# B&R Automation Studio project TD52 (part 38)

#### AdditionalFunctions.st - Additional functions
```iecst
(*******************************************************************************
coupling        additional functions

This code is confidential and proprietary to the INNIO Company.
It may not be used in any form, or reproduced in any manner,
without written permission of the INNIO Company.
Copyright, INNIO Company, 2019

Customized modifications: -
------------------------

History:
-------
V0.00.0	17.07.2012	froehlichw	new
V0.00.1	14.01.2019	Denk		adapted for bus test forcing

Instructions for use:
--------------------

Outstandings:
------------

(*******************************************************************************)

(*-----------------------------------------------------------------
/* compress and copy BOOL-Array at scrAdr to INT-Array at dstAdr
/* IN: scrAdr ... source address (start address of BOOL-Array)
/*     dstAdr ... destination address (base address=[0] of INT-Array)
/*     idxMin ... start index of INT-Array for copy
/*     idxMax ... end index of INT-Array for copy
/*---------------------------------------------------------------*)
ACTION BusTest_BOOL_TO_INT:
	FOR idx1:= idxMin TO idxMax DO
		pScrData ACCESS (srcAdr + (idx1 - idxMin) * 16);
		pDstData ACCESS (dstAdr + SIZEOF(pDstData) * idx1);
		pDstData.0:= pScrData[0];
		pDstData.1:= pScrData[1];
		pDstData.2:= pScrData[2];
		pDstData.3:= pScrData[3];
		pDstData.4:= pScrData[4];
		pDstData.5:= pScrData[5];
		pDstData.6:= pScrData[6];
		pDstData.7:= pScrData[7];
		pDstData.8:= pScrData[8];
		pDstData.9:= pScrData[9];
		pDstData.10:= pScrData[10];
		pDstData.11:= pScrData[11];
		pDstData.12:= pScrData[12];
		pDstData.13:= pScrData[13];
		pDstData.14:= pScrData[14];
		pDstData.15:= pScrData[15];
	END_FOR;
END_ACTION

(*-----------------------------------------------------------------
/* compress AND copy INT-Array at srcAdr TO BOOL-Array at dstAdr
/* IN: dstAdr ... destination address (start address OF BOOL-Array)
/*     scrAdr ... source address (base address=[0] OF INT-Array)
/*     idxMin ... start index OF INT-Array FOR copy
/*     idxMax ... end index OF INT-Array FOR copy
/*---------------------------------------------------------------*)
ACTION BusTest_INT_TO_BOOL:
	FOR idx1:= idxMin TO idxMax DO
		pScrData1 ACCESS (srcAdr + SIZEOF(pScrData1) * idx1);
		pDstData1 ACCESS (dstAdr + (idx1 - idxMin) * 16);
		pDstData1[0]:= pScrData1.0;
		pDstData1[1]:= pScrData1.1;
		pDstData1[2]:= pScrData1.2;
		pDstData1[3]:= pScrData1.3;
		pDstData1[4]:= pScrData1.4;
		pDstData1[5]:= pScrData1.5;
		pDstData1[6]:= pScrData1.6;
		pDstData1[7]:= pScrData1.7;
		pDstData1[8]:= pScrData1.8;
		pDstData1[9]:= pScrData1.9;
		pDstData1[10]:= pScrData1.10;
		pDstData1[11]:= pScrData1.11;
		pDstData1[12]:= pScrData1.12;
		pDstData1[13]:= pScrData1.13;
		pDstData1[14]:= pScrData1.14;
		pDstData1[15]:= pScrData1.15;
	END_FOR;
END_ACTION
```

#### coupling.var - Local variables
```iecst
VAR
	ucTeilerLauf : USINT; (* TK4 splitter variable *)
	ucINIT : ARRAY[0..1] OF USINT; (* initialise all coupling types *)
	szMode1 : STRING[50]; (* string interface mode 1 *)
	szInterface05 : STRING[40]; (* string interface 5 *)
	szInterface04 : STRING[40]; (* string interface 4 *)
	szInterface03 : STRING[40]; (* string interface 3 *)
	szInterface02_Comm2 : STRING[40]; (*Profibus communication2, slave2 *)
	szInterface02_Comm1 : STRING[40]; (*Profibus communication1, slave2 *)
	szInterface02 : STRING[40]; (* string interface 2 *)
	szInterface01_Comm2_PN : STRING[40]; (*Profinet communication2, slave1*)
	szInterface01_Comm2 : STRING[40]; (*Profibus communication2, slave1 *)
	szInterface01_Comm1_PN : STRING[40]; (*Profinet communication1, slave1 *)
	szInterface01_Comm1 : STRING[40]; (*Profibus communication1, slave1 *)
	szInterface01 : STRING[40]; (* string interface 1 *)
	szHilf1 : STRING[50]; (* help sting 1 *)
	szDevice1 : STRING[40]; (* string interface position 1 *)
	StationNumber : STRING[3];
	StationName1 : STRING[30] := ''; (*Profinet communication 1, station name*)
	Station : UDINT;
	Start_PN_Slave1 : USINT; (*Index variable*)
	Start_PB_Slave2 : USINT; (*Index variable*)
	Start_PB_Slave1 : USINT; (*Index variable*)
	siComm2_type : INT; (* couple type 2 old *)
	siComm2_Stopbit : INT; (* stop bits old Modbus *)
	siComm2_SlaveID : INT; (* ident for Modbus connection *)
	siComm2_Parity : INT; (* parity old Modbus *)
	siComm2_Interface : INT; (* position interface coupling 2 *)
	siComm2_Baud : INT; (* baudrate old Modbus *)
	siComm1_type : INT; (* couple type 1 old *)
	siComm1_Stopbit : INT; (* stop bits old Modbus *)
	siComm1_SlaveID : INT; (* ident for Modbus connection *)
	siComm1_Parity : INT; (* parity old Modbus *)
	siComm1_Interface : INT; (* position interface coupling 1 *)
	siComm1_Baud : INT; (* baudrate old Modbus *)
	nxpnsStartBusComm_01 : nxpnsStartBusComm;
	nxpnsSetName_01 : nxpnsSetName;
	nxdpsStartBusComm_02 : nxdpsStartBusComm;
	nxdpsStartBusComm_01 : nxdpsStartBusComm;
	nxdpsSetAdr_02 : nxdpsSetAdr;
	nxdpsSetAdr_01 : nxdpsSetAdr;
	MBT_4_2 : ARRAY[0..MODBUS_TCP_MAX_ARRAY] OF UINT := [MODBUS_TCP_MAX_ARRAY+1(0)]; (* data array Modbus TCP Coupling 2*)
	MBT_4_1 : ARRAY[0..MODBUS_TCP_MAX_ARRAY] OF UINT := [MODBUS_TCP_MAX_ARRAY+1(0)]; (* data array Modbus TCP Coupling 1*)
	MBSOpen_Var : ARRAY[0..1] OF MBSOpen; (* FUB Modbus open *)
	MBSlave_Var : ARRAY[0..1] OF MBSlave; (* FUB Modbus slave *)
	MBSClose_Var : ARRAY[0..1] OF MBSClose; (* FUB Modbus close *)
	MBR_4_2 : ARRAY[0..MODBUS_RTU_MAX_ARRAY] OF UINT := [MODBUS_RTU_MAX_ARRAY+1(0)]; (* data array Modbus RTU coupling 2 *)
	MBR_4_1 : ARRAY[0..MODBUS_RTU_MAX_ARRAY] OF UINT := [MODBUS_RTU_MAX_ARRAY+1(0)]; (* data array Modbus RTU coupling 1 *)
	MBinitOK : ARRAY[0..1] OF BOOL; (* initialising Modbus O.K. *)
	logErrorStringPN : STRING[100] := 'Error PROFINET communication slave 1';
	logErrorString2 : STRING[100] := 'Error PROFIBUS communication slave 2';
	logErrorStringModTCP : STRING[100] := 'Error MODBUS TCP set IP adress / Subnet mask slave';
	logErrorString1 : STRING[100] := 'Error PROFIBUS communication slave 1';
END_VAR
VAR CONSTANT
	IF4_IDLE : UINT := 0; (*Set IP adress and subnet mask IF4.ETH*)
	IP_IF4_SET : UINT := 1; (*Set IP adress IF4.ETH*)
	SUBMASK_IF4_SET : UINT := 2; (*Set Subnet mask IF4.ETH*)
	IF4_OK : UINT := 3; (*Set IP adress and subnet mask IF4.ETH OK*)
	OPEN_MODTCP : UINT := 4; (*Open Modbus TCP Communication*)
	IF4_ERR : UINT := 5; (*Set IP adress IF4.ETH Error*)
	PROFIBUS_MAX_RECV_2SLAVES : UINT := 16; (* max send data words profibus *)
	PROFIBUS_MAX_SEND_2SLAVES : UINT := 192; (* max send data words profibus *)
END_VAR
VAR
	iInterface02_Comm1 : UDINT; (*Adress Profibus Interface1, communication1, slave2*)
	iInterface01_Comm1_PN : UDINT; (*Adress Profinet Interface1, communication1, slave1*)
	iInterface01_Comm1 : UDINT; (*Adress Profibus Interface1, communication1, slave1 *)
	idx : INT;
	iComm1_PN_SlaveID1_old : INT; (*Profinet communication1, slave1 old adress*)
	iComm2_PN_SlaveID1_old : INT; (*Profinet communication1, slave1 old adress*)
	iComm1_PB_SlaveID1_old : INT; (*Profibus communication1, slave1 old adress*)
	iComm1_PB_SlaveID2_old : INT; (*Profibus communication1, slave2 old adress*)
	iComm2_PB_SlaveID1_old : INT; (*Profibus communication1, slave1 old adress*)
	iComm2_PB_SlaveID2_old : INT; (*Profibus communication1, slave2 old adress*)
	iComm_PB_SlaveID1 : INT; (*Profibus communication1, slave1 old adress*)
	iComm_PB_SlaveID2 : INT; (*Profibus communication1, slave1 old adress*)
	iComm_PN_SlaveID1 : INT; (*Profibus communication1, slave1 old adress*)
	AsArLogWrite_PN_01 : AsArLogWrite;
	AsArLogWrite_PB_02 : AsArLogWrite;
	AsArLogWrite_TCP : AsArLogWrite;
	AsArLogWrite_PB_01 : AsArLogWrite;
	AsArLogGetInfo_PN_01 : AsArLogGetInfo;
	AsArLogGetInfo_PB_02 : AsArLogGetInfo;
	AsArLogGetInfo_TCP : AsArLogGetInfo;
	AsArLogGetInfo_PB_01 : AsArLogGetInfo;
	InDataSwap : ARRAY[0..MAX_IN_DATA_ARRAY] OF INT;
	OutDataSwap : ARRAY[0..MAX_OUT_DATA_ARRAY] OF INT;
	OutDataOldSwap : ARRAY[0..MAX_OUT_DATA_ARRAY] OF INT;
	ArrayCntIn : INT;
	ArrayCntOut : INT;
	iStartRecvReg : INT;
	iStartRecvReg_old : INT;
	iStartSendReg : INT;
	iStartSendReg_old : INT;
	iIdx_Comm1_type_old : INT; (*Type of coupling 1 old, for detection of parameter change*)
	iIdx_Comm2_type_old : INT; (*Type of coupling 2 old, for detection of parameter change*)
	iBC_Test_Recv_Reg_old : ARRAY[0..MAX_IN_DATA_ARRAY_BUSTEST] OF INT;
	bBC_Test_Recv_Reg_old : ARRAY[0..MAX_IN_DATA_ARRAY_BOOL] OF BOOL;
	idx1 : INT;
	srcAdr : UDINT;
	dstAdr : UDINT;
	idxMin : INT;
	idxMax : INT;
	pScrData : REFERENCE TO ARRAY[0..15] OF BOOL;
	pDstData : REFERENCE TO UINT;
	pScrData1 : REFERENCE TO UINT;
	pDstData1 : REFERENCE TO ARRAY[0..15] OF BOOL;
	RegOffset_Send : INT;
	RegOffset_Recv : INT;
	xTON_BC_Test_Force_Active : TON;
	bBC_Test_Recv_Reg_Forced : ARRAY[0..MAX_IN_DATA_ARRAY] OF BOOL;
	bBC_Test_Send_Reg_Forced : ARRAY[0..MAX_OUT_DATA_ARRAY] OF BOOL;
	iBC_Test_Recv_Start_Reg_old : INT;
	iBC_Test_Send_Start_Reg_old : INT;
	bBC_Test_Recv_Reg_Forced_old : ARRAY[0..20] OF BOOL;
	bBC_Test_Send_Reg_Forced_old : ARRAY[0..20] OF BOOL;
	bBC_Test_Recv_Reg_AllForced : BOOL;
	bBC_Test_Send_Reg_AllForced : BOOL;
	bBC_Test_Recv_Reg_AllUnforced : BOOL;
	bBC_Test_Send_Reg_AllUnforced : BOOL;
	bBC_Test_Send_DW : BOOL; (*Dataword convention for send (Profibus, Profinet)*)
	iBC_Test_Send_DW : INT; (*Dataword convention for send (Profibus, Profinet)*)
	bBC_Test_Recv_DW : BOOL; (*Dataword convention for receive (Profibus, Profinet)*)
	iBC_Test_Recv_DW : INT; (*Dataword convention for receive (Profibus, Profinet)*)
	r : INT;
	i : INT;
	k : INT;
	t : INT;
	m : INT;
	n : INT;
	p : INT;
	v : INT;
	w : INT;
	x : INT;
	b : INT;
	iBC_Test_Send_Reg_old : ARRAY[0..MAX_OUT_DATA_ARRAY] OF INT;
	bBC_Test_Send_Reg_old : ARRAY[0..MAX_OUT_DATA_ARRAY_BOOL] OF BOOL;
	xTON_AutoToggle1 : TON;
	xTON_AutoToggle2 : TON;
	xTON_CustomToggle1 : TON;
	xTON_CustomToggle2 : TON;
	y : INT;
END_VAR
(* Modbus TCP General *)
VAR
	szComm_Device_TCP : STRING[20]; (*Device adress Modbus TCP slave (IF4.ETH)*)
	szComm_Device2_TCP : STRING[20]; (*Device adress Modbus TCP slave (IF4.ETH)*)
	szComm_Device3_TCP : STRING[20]; (*Device adress Modbus TCP slave (IF4.ETH)*)
	IP_ModTCP : UINT; (*Set IP adress IF4.ETH*)
END_VAR
(* Modbus TCP Coupling 1 *)
VAR
	iComm_Device_TCP : UDINT; (*Device adress Modbus TCP slave (IF4.ETH)*)
	iComm_SubMask_TCP : UDINT; (*Subnet mask Modbus TCP slave *)
	iComm_IPaddr_TCP : UDINT; (*IP adress Modbus TCP slave *)
	szComm_IPaddr_TCP_temp : STRING[20]; (*IP adress Modbus TCP slave *)
	szComm_IPaddr_TCP : STRING[20]; (*IP adress Modbus TCP slave *)
	szIPAddr1 : STRING[3]; (*temp for setting Modbus TCP IP adress*)
	szIPAddr2 : STRING[3]; (*temp for setting Modbus TCP IP adress*)
	szIPAddr3 : STRING[3]; (*temp for setting Modbus TCP IP adress*)
	szIPAddr4 : STRING[3]; (*temp for setting Modbus TCP IP adress*)
	szComm_SubMask_TCP_temp : STRING[20]; (*Subnet mask Modbus TCP slave *)
	szComm_SubMask_TCP : STRING[20]; (*Subnet mask Modbus TCP slave *)
	szSubMask3 : STRING[3]; (*temp for setting Modbus TCP Subnet mask*)
	szSubMask4 : STRING[3]; (*temp for setting Modbus TCP Subnet mask*)
	szSubMask1 : STRING[3]; (*temp for setting Modbus TCP Subnet mask*)
	szSubMask2 : STRING[3]; (*temp for setting Modbus TCP Subnet mask*)
	siComm_PortID_TCP : INT; (* ident for Modbus TCP connection *)
	siComm_SlaveID_TCP : INT; (* ident for Modbus TCP connection *)
	ucINIT_IP_addr_TCP : USINT;
	fMBTSOpen_Var : fMBTSOpen; (* FUB Modbus TCP slave open *)
	fMBTSClose_Var : fMBTSClose; (* FUB Modbus TCP slave close *)
	CfgSetSubnetMask_01 : CfgSetSubnetMask; (*FUB Subnet Mask Config*)
	CfgSetIPAddr_01 : CfgSetIPAddr; (*FUB IP Config*)
	bMBtcpinit : ARRAY[0..1] OF BOOL; (* initialise Modbus TCP *)
	bMBinit : ARRAY[0..1] OF BOOL; (* initialise Modbus *)
END_VAR
(* Modbus TCP Coupling 2*)
VAR
	iComm2_Device_TCP : UDINT; (*Device adress Modbus TCP slave (IF4.ETH)*)
	iComm2_SubMask_TCP : UDINT; (*Subnet mask Modbus TCP slave *)
	iComm2_IPaddr_TCP : UDINT; (*IP adress Modbus TCP slave *)
	szComm2_IPaddr_TCP_temp : STRING[20]; (*IP adress Modbus TCP slave *)
	szComm2_IPaddr_TCP : STRING[20]; (*IP adress Modbus TCP slave *)
	szComm2_IPAddr1 : STRING[3]; (*temp for setting Modbus TCP IP adress*)
	szComm2_IPAddr2 : STRING[3]; (*temp for setting Modbus TCP IP adress*)
	szComm2_IPAddr3 : STRING[3]; (*temp for setting Modbus TCP IP adress*)
	szComm2_IPAddr4 : STRING[3]; (*temp for setting Modbus TCP IP adress*)
	szComm2_SubMask_TCP_temp : STRING[20]; (*Subnet mask Modbus TCP slave *)
	szComm2_SubMask_TCP : STRING[20]; (*Subnet mask Modbus TCP slave *)
	szComm2_SubMask3 : STRING[3]; (*temp for setting Modbus TCP Subnet mask*)
	szComm2_SubMask4 : STRING[3]; (*temp for setting Modbus TCP Subnet mask*)
	szComm2_SubMask1 : STRING[3]; (*temp for setting Modbus TCP Subnet mask*)
	szComm2_SubMask2 : STRING[3]; (*temp for setting Modbus TCP Subnet mask*)
	siComm2_PortID_TCP : INT; (* ident for Modbus TCP connection *)
	siComm2_SlaveID_TCP : INT; (* ident for Modbus TCP connection *)
	ucINIT_IP_addr_TCP2 : USINT;
	IP_ModTCP2 : UINT;
	fMBTSOpen2_Var : fMBTSOpen; (*FUB Modbus TCP Slave Open*)
	fMBTSClose2_Var : fMBTSClose; (*FUB Modbus TCP Slave Close*)
	fMBTSlave2_Var : fMBTSlave; (*FUB Modbus TCP Slave*)
	CfgSetSubnetMask_02 : CfgSetSubnetMask; (*FUB Subnet Mask Config*)
	CfgSetIPAddr_02 : CfgSetIPAddr; (*FUB IP Config*)
END_VAR
```

### Program Logical/Coupling/MBRMaster (IEC, version 4.12.0) - Modbus RTU Master

#### MBRMaster.st - Implementation code
```iecst
(*******************************************************************************
Coupling:    Modbus RTU Master

This code is confidential and proprietary to the INNIO Company.
It may not be used in any form, or reproduced in any manner,
without written permission of the INNIO Company.
Copyright, INNIO Company, 2019

Customized modifications: -
------------------------

History:
-------
V04.05.00	22.07.2017	Denk		new
V04.12.00	29.03.2023	Denk		Device adress changed

Instructions for use:
--------------------
Modbus RTU Master <--> SCR HUG Smart Dosing Box Slave
SCR logic in Emission module
Possible Slave#2 prepared

Outstandings:
------------

(*******************************************************************************)

PROGRAM _INIT

	(* EDIT: Adress *)
	device:= 'SL2.IF1.ST66.IF1.ST2.IF1';

	(* EDIT: PHY = Physical | PA = Parity | SB = Stopbit | BD = Baudrate *)
	mode:= '/PHY=RS485 /PA=N /DB=8 /SB=1 /BD=9600';

	(* EDIT: Config file for slave adress,register, function code, ... *)
	config:= 'cfg_mbus';

	timeout:= 300;

	stepMbMaster:= stpMbM_WAIT;
	cmdMbMOpen:= TRUE;

	(* EDIT: IN/OUT data register *)
	MBM_SCR_Register[0];				(* Slave SCR *)
//	MBM_FieldDevice1_Register[0];		(* Slave 2, CEMS*)

	(* EDIT: IN/OUT data interfaces *)
	OUT_CP.iModbus_SCR_UINT;			(* Slave SCR *)
	OUT_CP.iModbus_SCR_INT;		 		(* Slave SCR, for INT register 73,74,75*)
	IN_CP.iModbus_SCR;					(* Slave SCR *)
//	OUT_CP.iMBM_FieldDevice1_Receive;	(* Slave 2, CEMS *)
//	IN_CP.iMBM_FieldDevice1_Send;		(* Slave 2, CEMS *)

END_PROGRAM

PROGRAM _CYCLIC
IF ucTeilerLauf > ucTeilerMaster THEN
	CASE stepMbMaster OF
	  (*----------------------------------------------------------
	  /* wait
	  /*---------------------------------------------------------*)
		stpMbM_WAIT:
			IF cmdMbMOpen THEN
				cmdMbMOpen:= FALSE;
				stepMbMaster:= stpMbM_OPEN;
			END_IF;

	  (*----------------------------------------------------------
	  /* open device
	  /*---------------------------------------------------------*)
		stpMbM_OPEN:
			MBMOpen_0.enable:= TRUE;
			MBMOpen_0.pDevice:= ADR(device);
			MBMOpen_0.pMode:= ADR(mode);
			MBMOpen_0.pConfig:= ADR(config);
			MBMOpen_0.timeout:= timeout;
			MBMOpen_0.ascii:= 0;
			MBMOpen_0();
			IF (MBMOpen_0.status <> ERR_FUB_BUSY) THEN
				IF (MBMOpen_0.status = ERR_OK) THEN
					MBMaster_0.enable:= TRUE;
					MBMaster_0.ident:= MBMOpen_0.ident;
					stepMbMaster:= stpMbM_RUN;
				ELSE
					stepMbMaster:= stpMbM_ERROR;
				END_IF;
			END_IF;

	  (*----------------------------------------------------------
	  /* run master
	  /*---------------------------------------------------------*)
		stpMbM_RUN:
			IF cmdMbMClose THEN
				cmdMbMClose:= FALSE;
				MBMaster_0.enable:= FALSE;
				MBMClose_0.enable:= TRUE;
				MBMClose_0.ident:= MBMOpen_0.ident;
				stepMbMaster:= stpMbM_CLOSE;
			END_IF;

			MBMaster_0();

			(* Slave SCR *)
			memcpy(ADR(MBM_SCR_Register_swapped[65]), ADR(MBM_SCR_Register[65]), 16);	 		//Register Offset Anpassung hier: MBM_SCR_Register[xx]
			FOR ArrayCntOut := 65 TO 69 BY 1 DO
				OUT_CP.iModbus_SCR_UINT[ArrayCntOut] := (*swapINT*)(MBM_SCR_Register_swapped[ArrayCntOut]);
			END_FOR;
			FOR ArrayCntOut := 70 TO 72 BY 1 DO
				OUT_CP.iModbus_SCR_UINT[ArrayCntOut] := (*swapINT*)(MBM_SCR_Register_swapped[ArrayCntOut]);
			END_FOR;

			memcpy(ADR(MBM_SCR_Register_swapped73[73]), ADR(MBM_SCR_Register[73]), 6);
			FOR ArrayCntOut := 73 TO 75 BY 1 DO
				OUT_CP.iModbus_SCR_INT[ArrayCntOut] := (*swapINT*)(MBM_SCR_Register_swapped73[ArrayCntOut]);
			END_FOR;

			memcpy(ADR(MBM_SCR_Register_swapped[76]), ADR(MBM_SCR_Register[76]), 18);
			FOR ArrayCntOut := 76 TO 84 BY 1 DO
				OUT_CP.iModbus_SCR_UINT[ArrayCntOut] := (*swapINT*)(MBM_SCR_Register_swapped[ArrayCntOut]);
			END_FOR;

			memcpy(ADR(MBM_SCR_Register_swapped[1]), ADR(IN_CP.iModbus_SCR[1]), 1);
			FOR ArrayCntIn := 1 TO 1 BY 1 DO
				MBM_SCR_Register[ArrayCntIn] := (*swapINT*)(MBM_SCR_Register_swapped[ArrayCntIn]);
			END_FOR;

			memcpy(ADR(MBM_SCR_Register_swapped[2]), ADR(IN_CP.iModbus_SCR[2]), 19);
			FOR ArrayCntIn := 2 TO 20 BY 1 DO
				MBM_SCR_Register[ArrayCntIn] := (*swapINT*)(MBM_SCR_Register_swapped[ArrayCntIn]);
			END_FOR;

//			(* Slave 2, CEMS *)
//			memcpy(ADR(OUT_CP.iMBM_FieldDevice1_Receive[0]), ADR(MBM_FieldDevice1_Register[0]), MODBUS_RTU_MASTER_MAX_ARRAY);
//			memcpy(ADR(MBM_FieldDevice1_Register[200]), ADR(IN_CP.iMBM_FieldDevice1_Send[0]), MODBUS_RTU_MASTER_MAX_ARRAY);

			(* cyclic read and write *)
			(* function code 03 read holding registers *)
			(* function code 16 write multiple registers *)
			(* Slave SCR *)
			IF Para.bSCR_BUS_Exist THEN
				EvReadMBR_SCR := TRUE;
			END_IF;
			IF Para.bSCR_BUS_Exist THEN
				EvWriteMBR_SCR := TRUE;
			END_IF;

//			(* Slave 2, CEMS *)
//			IF (EvReadMBR_4_1_1 = FALSE) THEN
//				EvReadMBR_4_1_1 := TRUE;
//			END_IF;
//			IF (EvWriteMBR_4_1 = FALSE) THEN
//				EvWriteMBR_4_1 := TRUE;
//			END_IF;

	  (*----------------------------------------------------------
	  /* close device
	  /*---------------------------------------------------------*)
		stpMbM_CLOSE:
			MBMClose_0();
			IF (MBMClose_0.status <> ERR_FUB_BUSY) THEN
				IF (MBMClose_0.status = ERR_OK) THEN
					stepMbMaster:= stpMbM_WAIT;
				ELSE
					stepMbMaster:= stpMbM_ERROR;
				END_IF;
			END_IF;

	  (*----------------------------------------------------------
	  /* error
	  /*---------------------------------------------------------*)
		stpMbM_ERROR:
			IF cmdMbMQuitError THEN
				cmdMbMQuitError:= FALSE;
				stepMbMaster:= stpMbM_WAIT;
			END_IF;

	END_CASE;

END_IF;

IF ucTeilerLauf > ucTeilerMaster THEN
	ucTeilerLauf:= 0;
END_IF;
ucTeilerLauf:= ucTeilerLauf + 1;

END_PROGRAM
```

#### MBRMaster.var - Local variables
```iecst
VAR
	device : STRING[40];
	mode : STRING[40];
	config : STRING[40];
	timeout : UINT;
	stepMbMaster : stepMbMasterEnum;
	cmdMbMOpen : BOOL;
	cmdMbMClose : BOOL;
	cmdMbMQuitError : BOOL;
	MBMOpen_0 : MBMOpen;
	MBMaster_0 : MBMaster;
	MBMClose_0 : MBMClose;
	EvReadMBR_SCR : BOOL;
	EvWriteMBR_SCR : BOOL;
	ucTeilerMaster : INT := 20;
	ucTeilerLauf : INT;
	ArrayCntOut : INT;
	ArrayCntIn : INT;
END_VAR
```

#### MBRMaster.typ - Local data types
```iecst
TYPE
	stepMbMasterEnum :
		(
		stpMbM_WAIT,
		stpMbM_OPEN,
		stpMbM_RUN,
		stpMbM_CLOSE,
		stpMbM_ERROR
		);
END_TYPE
```

### Data object Logical/Coupling/cfg_mbus (Simple, version 4.05.0)

#### cfg_mbus.dat
```
(*******************************************************************************
Coupling:    Modbus RTU Master query configuration

This code is confidential and proprietary to the INNIO Company.
It may not be used in any form, or reproduced in any manner,
without written permission of the INNIO Company.
Copyright, INNIO Company, 2019

Customized modifications: -
------------------------

History:
-------
V04.05.00	22.07.2017	Denk		new

Instructions for use:
--------------------
Modbus RTU Master <--> SCR HUG Smart Dosing Box Slave
Register query configuration
Possible Slave#2 prepared

Outstandings:
------------

*******************************************************************************)
; Structure of entry
; ------------------
; "EventPV1 ", 01, $01, "LocalPV1 ", 0000, 0005
;     |        |    |       |         |     |
;     |        |    |       |         |     +--- data lenght
;     |        |    |       |         +--------- data offsset
;     |        |    |       +------------------- scr/dest PV
;     |        |    +--------------------------- destination ID
;     |        +-------------------------------- function code
;     +----------------------------------------- event PV

;--------------------
; Modbus command file
;--------------------

"MBRMaster:EvReadMBR_SCR", 03, $01, "MBRMaster:MBM_SCR_Register[65]",  0064, 0020,
"MBRMaster:EvWriteMBR_SCR",  16, $01, "MBRMaster:MBM_SCR_Register[1]", 0000, 0010,

(*"MBRMaster:EvReadMBR_4_1_1", 03, $06, "MBRMaster:MBM_FieldDevice1_Register[0]",   0000, 0016,
"MBRMaster:EvWriteMBR_4_1",  16, $06, "MBRMaster:MBM_FieldDevice1_Register[200]", 0016, 0016*)
```

### Program Logical/Coupling/ParCP (IEC, version 4.06.0) - + Parameter handling

- perm_par.st (not readable text: treated as protected, skipped)

#### perm_par.var
```iecst
VAR
	tParaIntern : ParaHandler_typ; (*Connector type to perm_par*)
	tMM2ParaBase_ReadBack : MM2ParaBase_type; (*INTERNAL! V4.06 new readback structure for information from previous tasks*)
	bWriteDataObj : BOOL; (* TRUE=write data object module *)
	bDataObjLenErr : BOOL; (*Error occured in permem: data module size missmatch*)
	bCreateDataObj : BOOL; (* TRUE=create new data object *)
	bWriteOnce : BOOL; (* write permanent memory once *)
	DatObjCreate_01 : DatObjCreate; (* data object create *)
	DatObjInfoBak_02 : DatObjInfo; (* data object info *)
	DatObjDelete_01 : DatObjDelete; (* data object delete *)
	DatObjRead_01 : DatObjRead; (* data object read *)
	DatObjRead_02 : DatObjRead; (* manual initiated data object read *)
	DatObjWrite_01 : DatObjWrite; (* data object write *)
	DatObjDelete_02 : DatObjDelete; (* data object delete *)
	DatObjDelete_11 : DatObjDelete; (*Delete Backup File*)
	DatObjInfo_01 : DatObjInfo; (* data object info *)
	DatObjInfo_02 : DatObjInfo; (* data object info *)
	szModuleName : STRING[35]; (* module name of object *)
	szModuleNameBackup : STRING[35]; (* module name of posiibly created backup object *)
	DatObjCopy_01 : DatObjCopy;
	bCopyDataObj : BOOL;
	TON_WarnDelay : TON;
	TON_WritePMEM : TON; (* delay write permanent memory *)
	ulPMPointer : UDINT; (* adress of actual checksum value *)
	ulChecksum : UDINT; (* parameter checksum value *)
	pm_len : UDINT; (* permanent value lenght *)
	ulChecksumOld : UDINT; (* last vlaue of parameter checksum *)
	ulChkValue : UDINT; (* actual value of parameter pointer *)
	pm_id : UDINT; (* permanent value identifier *)
	pm_p : UDINT; (* permanent value pointer *)
	DatObjInfo_META : DatObjInfo;
	DatObjRead_META : DatObjRead;
	szMetaDataRaw : STRING[2000];
	szMetaData : ARRAY[0..4] OF STRING[35];
	szMetaDataVis : ARRAY[0..3] OF STRING[35];
	ssIndex : INT;
	ssCount : INT;
	ucMetaDataRaw : ARRAY[0..2000] OF USINT;
	ssCount2 : INT;
	szMetaDataFile : STRING[10];
	szText1 : STRING[20];
	pv_adr_IN_XX_tPB2MM : UDINT;
	pv_lng : UDINT;
	pv_lng_IN_XX_tPB2MM : UDINT;
	pv_lng_OUT_XX_tPB2MM : UDINT;
	szText2 : STRING[20];
	pv_adr_OUT_XX_tXX2PB : UDINT;
END_VAR
VAR CONSTANT
	ERR_NOERROR : UINT := 0;
END_VAR
VAR
	usPMWriteCnt : UINT;
	pm_Error : UDINT; (* permanent value error *) (* Deleted: pm : ParaMem_typ; permanent memory tags mathias, 22.8.11*)
	fun_Error : UDINT := 0; (*state > 0 = function error*)
	xLocalParaCheck : ParaCheckFUB; (*local function instance to check parameter values*)
	TON_ParaSetupOk : TON;
	bParaCheckSystemOk : BOOL;
	iDebug_ParaOkChecked : UDINT;
	bRestoreBackupDataObj : BOOL := FALSE;
	bRestoreDataObjContent : BOOL := FALSE;
	pm_id_backup : UDINT;
	pm_p_Backup : UDINT;
	DatObjCopy_02 : DatObjCopy;
	bDeleteBackupDataObj : BOOL := FALSE; (*Command to delete backup data module file on purpose*)
	bDebugPara : ARRAY[0..5] OF BOOL;
	ssIndex2 : INT;
	ssIndex3 : INT;
	ssIndex4 : INT;
	ssIndexVis : INT;
	szText : STRING[40];
	pv_adr_Para : UDINT;
	szParaSnippet : ARRAY[0..5] OF STRING[150];
	szParaIndex : STRING[10];
	slValue : DINT;
	iModuleDLD_ResetCount : INT;
	bDownloadDetected : BOOL;
	bFlagParaStructCopyWorking : BOOL; (*true, if cyclic para copying is active, 1 false cycle at every copy *)
	bStoreInitParaInDataObj : BOOL := FALSE;
	bTestflag : BOOL;
	bReadOutMETA_Once : BOOL;
	tParaCheck_iPvAdress : ARRAY[0..5] OF UDINT;
	tParaCheck_iPvLengt : ARRAY[0..5] OF UDINT;
	tParaCheck_rPvValue : ARRAY[0..5] OF REAL;
	tParaCheck_rRangeMIN : ARRAY[0..5] OF REAL;
	tParaCheck_rRangeMAX : ARRAY[0..5] OF REAL;
	tParaCheck_szPvName : ARRAY[0..5] OF STRING[35];
	ssFormatDetected : INT;
	szMetaDataPart : STRING[150];
	szFullTaskName : STRING[35];
	szFullMetaModuleName : STRING[35];
	debugLen : INT;
	debugSize : INT := 0;
	strcat_adr1 : UDINT;
	strcat_adr2 : UDINT;
	ssIndexTN : INT;
	bAlternate : BOOL;
	n : INT;
	iAlternateChecksum : DINT;
	iAlternateChecksumOld : DINT;
	ulDebugChkValue : ARRAY[0..999] OF UDINT;
	Adr1 : UDINT;
	Adr2 : UDINT;
	usPMWriteCntStepsize : UINT := 1; (*different step sizes to help debug*)
	usPMWriteCntXOR : UINT;
	usPMWriteCntAltSum : UINT;
	ulAdrPM : UDINT;
	usChkValuePM : USINT;
	ulAdrPara : UDINT;
	ulPara_len : UDINT;
	usChkValuePara : USINT;
	iDebugCountPMDifferences : DINT := 0;
	bEngineRunDetected : BOOL; (*detection status bit autocommand 100 /101  for engine run state*)
	ucMetaDataDebugInfoLine : ARRAY[0..24] OF STRING[80];
	ssIndexMand : INT := 0;
	szMetaDataMand : STRING[35];
	iMyErrorInfo_Autoreset : DINT; (*internal autoreset counter*)
	ssIndex_Version : INT; (*internal*)
	ssIndex_BU : INT; (*internal*)
	ssIndex_BU2 : INT; (*internal*)
END_VAR
```

### Program Logical/Coupling/MsgCP (IEC, version 4.05.0) - + Messages

- MsgCPCyclic.st (not readable text: treated as protected, skipped)

- MsgCPInit.st (not readable text: treated as protected, skipped)

#### MsgCP.var
```iecst
VAR
	iAdrAmmBase2MM : UDINT;
	iAdrMM2AmmBase : UDINT;
	xMsg1151 : Msg;
	xMsg1150 : Msg;
	xMsg1099 : Msg;
	xMsg1147 : Msg;
END_VAR
```

### Package Logical/Customized - CU: Customize

### Data object Logical/Customized/META_CU (Simple) - MODUL META data file

#### META_CU.dat
```
; *******************************************************************************
; AGGR: Module Meta Data (data module)
;
; This code is confidential and proprietary to the INNIO Company.
; It may not be used in any form, or reproduced in any manner, without the express
; written permission of the INNIO Company.
; Copyright, INNIO Company, 2023
;
; Customized modifications: -
; ------------------------
;
; History:
; -------
; V3.99		06-03-2013	Weitzer, generated for modular software
; V4.02.0	11.06.2015	Zengerer version + dependencies changed (IF change with array index 0 for compatibility with c-tasks)
; V4.03.00	02.11.2015	Zengerer MANDATORYMODULE
; V4.05.03	09.03.2018	Zengerer header cleared
;
; V4.25.00	28.01.2026	in THIS LINE HERE update ONLY version number and date; state changees below in INFO section;
;
; Instructions for use:
; --------------------
; make only changes at the version numbers
;
; Outstandings:
; ------------
;
;
; *******************************************************************************
;
"<META>"
;
; Module ID
"<MODUL>CU</MODUL>"
;
; Module Version (xx.yy.zz.cc)
"<VERSION>04.25.00.03</VERSION>"
;
; Module Basisupdate Version BU (00-99)
"<BASISUPDATE_VERSION>00</BASISUPDATE_VERSION>"

; Optional: specify order number for limitated module usage
"<ORDER>DT52</ORDER>" ;<!--(optional, wenn nicht vorhanden dann für alle Aufträge gültig)-->
;
; Parameter Check (Name:=aAbcdef; MIN:=xxx; MAX:=yyy;)
"<PARAMETER_CHK>"
"	<PARA1 Name='iEng_Motortype' MIN='208' MAX='1920' />"
"	<PARA2 Name='rN_EngStart_LimHi' MIN='50.0' MAX='2200.0' />"
"	<PARA3></PARA3>"
"	<PARA4></PARA4>"
"	<PARA5></PARA5>"
"</PARAMETER_CHK>"
;
; Statement, if engine operation is also allowed without this module (FALSE) or if this modules parameter check passing is mandatory (TRUE)
"<MANDATORYMODULE>FALSE</MANDATORYMODULE>"
;
; Permanent Datamodule Filenames<!-- state filename only, without extension; use e.g. for counter information storage-->
"<DATAMODULES>" ;<!-- optional more than 1 lines allowed. Do not state backup storage module p1BAK_CU here -->
"	<DATAMODULE>perm1_CU</DATAMODULE>"
"	<DATAMODULE>par_CU</DATAMODULE>"
"</DATAMODULES>"
;
; Dependencies Modules (MMxx.yy.zz.cc)
"<DEPENDENCIES>"
"	<DEPENDENCY MODULE='AB' VERSION='04.07.01.00' />" 	; Add dependencies for customization here
"	<DEPENDENCY MODULE='AG' VERSION='04.14.00.00' />"	; for new TC_CoolDownRun alarms 2015-02-23,
"	<DEPENDENCY MODULE='CH' VERSION='04.10.00.00' />"	; Add dependencies for customization here
"	<DEPENDENCY MODULE='CP' VERSION='04.13.00.00' />"	; ...
"	<DEPENDENCY MODULE='EC' VERSION='04.13.00.00' />"	;FastStart V4.06
"	<DEPENDENCY MODULE='EG' VERSION='04.04.00.00' />"	; ...
"	<DEPENDENCY MODULE='EM' VERSION='04.04.00.00' />"
"	<DEPENDENCY MODULE='EX' VERSION='04.10.00.00' />"
"	<DEPENDENCY MODULE='GC' VERSION='04.10.00.00' />"
"	<DEPENDENCY MODULE='GD' VERSION='04.04.00.00' />"
"	<DEPENDENCY MODULE='GM' VERSION='04.04.00.00' />"
"	<DEPENDENCY MODULE='GR' VERSION='04.13.00.00' />"
"	<DEPENDENCY MODULE='GT' VERSION='04.10.01.00' />"
"	<DEPENDENCY MODULE='HA' VERSION='04.14.00.00' />"
"	<DEPENDENCY MODULE='HC' VERSION='04.10.00.00' />" 	;rT_ChC_Ctr_Wex_Cust add V4.5 new interface...
"	<DEPENDENCY MODULE='IC' VERSION='04.04.00.00' />"
"	<DEPENDENCY MODULE='IG' VERSION='04.10.00.00' />"
"	<DEPENDENCY MODULE='KL' VERSION='04.04.00.00' />"
"	<DEPENDENCY MODULE='KN' VERSION='04.10.00.00' />"
"	<DEPENDENCY MODULE='MO' VERSION='04.04.00.00' />"
"	<DEPENDENCY MODULE='OP' VERSION='04.13.00.00' />"
"	<DEPENDENCY MODULE='PB' VERSION='04.06.00.00' />" 	;new permanent file info
"	<DEPENDENCY MODULE='SA' VERSION='04.04.00.00' />"
"	<DEPENDENCY MODULE='SY' VERSION='04.13.00.00' />"
"	<DEPENDENCY MODULE='TR' VERSION='04.10.00.00' />"
"	<DEPENDENCY MODULE='VE' VERSION='04.07.00.00' />"
"	<DEPENDENCY MODULE='VI' VERSION='04.09.00.00' />"
"   <DEPENDENCY VISVERSION='02.15.00.00' />"			; Dependencies Visualization
"</DEPENDENCIES>"
;
; Module function description
"<MODULEFUNCTION>" ;<!-- short overview documentation of module function; add reference to detailed information, if available-->
"	<General>	"
"	MM Customized is a collection of prepared spare items for individual adoptions. "
"	</General>	"
""
"	<F1 Name='Analog Inputs and Outputs' LastModified='4.0.0.0'>"
"	Predefined Channels (CustAnaIn[]) for plant specific purpose, usage defined hardcodede at time of sw generation.	"
"   Last Update: Separation of unchangeable code parts of tasks ran_def and MsgCU into new tasks in Cust_Internals"
"	</F1>"
"	<F2 Name='Digital Inputs and Outputs'  LastModified='4.0.0.0'>"
"	Predefined Channels (CustDigIn[]) for plant specific purpose, usage defined hardcodede at time of sw generation.	"
"	</F2>"
"	<F3 Name='Customizable controllers'  LastModified='4.0.0.0'>"
"	8 predefined PID- Controllers for plant specific purpose, usage defined hardcodede at time of sw generation.	"
"	</F3>"
"	<F4 Name='Customer Inputs and Outputs'  LastModified='4.0.0.0'>"
"	Prepared channels with highly parameter definable function for changeable Inputs and Outputs (CustomerIO), without hardcodeded purpose at time of sw generation.	"
"	</F4>"
"	<F5 Name='Customer Messages'  LastModified='4.2.2.0'>"
"	Additional 300 Messages prepared for : Alarms 1601-1700, Warnings 1701-1800, Operating messages 3601-3700, IN Interface cleanup	"
"	</F5>"
"	<F6 Name='Customer Counters'  LastModified='4.2.2.0'>"
"	New OUT Interface rCA_PI_Dur_COffset for custom PI duration offset "
"	10 Customizable Counters, stored in permanent memory file (last change 2015-02-04)	"
"	</F7>"
"	<F7 Name='Customizable Scaling Blocks'  LastModified='4.11.0.0'>"
"	10 predefined linear scaling blocks for plant specific purpose, usage defined hardcodede at time of sw generation.	"
"	</F7>"
""
"	<Info>"
"	This module is also the prefered place, where tasks to perform plant specific programmed functions are to be implemented.	"
"	Vis V2.02.x.x: Interface update prepared for reserve analog inputs, but still compatible with previous versions	"
"   UPDATE V4.2.0 version + dependencies changed (IF change with array index 0 for compatibility with c-tasks)	"
" 	UPDATE V4.2.2 cleanup, OPC handling part added for OPC DA values from VIS	"
"   UPDATE V4.3.0 version + dependencies changed (CAUSED BY ARRAY INDEX 0 for compatibility with c-tasks)	"
"   UPDATE V4.3.1 fix with ParaFactoryDefault for not jet released DO para	"
"   UPDATE V4.3.2 remove predefined reserve parameter numbers from task anf_nb to avoid unintended task activation  "
"   UPDATE V4.4.0 version + dependencies changed (CAUSED BY ARRAY SIZE INCREASE)	"
"   UPDATE V4.4.1 new task c_mns for standardized mains import controller (former task anf_nb retired)	"
"	UPDATE V4.4.2 task c_red replace IN_CU.tCustAnaIn[1].Ai by a neutral IN_CU.tCustAnaIn[0].Ai default "
"   UPDATE V4.4.3 module_CUPerm.typ keep length of perm with new iCount11-20"
"	UPDATE V4.4.4 rPr_Ch_P2s_Avg  IF625	bost pressure UNIT CHANGED to 1/100bar according to IF docu - Poppe Norber "
"	UPDATE V4.4.5 Connect In Interface to tP_Mns_AnaIn, tDem_Ctr_Mns"
"   UPDATE V4.4.6 update to frequency control"
"	UPDATE V4.4.7 30.06.2017	Gwiggner update to frequency control "
"	UPDATE V4.5.0 OUT_CU.rT_ChC_Ctr_Wex_Cust add new interface, clear bad interface vars "
"	UPDATE V4.5.0 Zengerer tDem_Ctr_Mns as enable condition for all AI alarms "
"	UPDATE V4.5.00 07.12.2017  Farre,   added/modified Q functions, Point of control/reference, P(U) "
"	UPDATE V4.5.00 04.12.2017	Messner	 bMsg1045, bMsg1069, bMsg1161, bMsg1162, bMsg1169, bMsg1170, bMsg1174, bMsg2112 deleted "
"	UPDATE V4.5.00 25.01.2018	Zengerer bParaSetupOk as enable condition for all AI alarms  "
"	UPDATE V4.5.01 22.02.2018	lettenb. AI_PF_CosPCtr_Set removed	"
"	BETA   V4.5.2 optional prepared customizable interface  - BETA PHASE, use only in coordination with TPSS"
"	UPDATE V4.5.4 Zengerer bParaSetupOk as enable condition for alarm 2302, 8966-, 3701-"
"	UPDATE V4.5.6 26.03.2018	Farre, Signals removed (PF_CosPCtr_PF1_Ena, PF_CosPCtr_PF2_Ena, PF_CosPCtr_PF3_Ena, PF_CosPCtr_PF4_Ena, PF_CosPCtr_PF5_Ena)"
"       		  13.04.2018	Zengerer comments for retired msg datapoints, no functional changes"
"	V4.05.06	  18.06.2018	Gwiggner BU 01: power setpoint for Next-Box hardwire"
"                 05.09.2018	Zuschnig BU 01: Added activation to use frozen signals for P_Set, P_Lim, COSPHI_Set, Q_Set, Q_Lim and U_Set "
"	UPDATE V4.7.0 09.08.2018	Schmid, 2nd low temperature charge cooling circuit added, change in tManAuxCtr struct"
"	V4.07.01.0 Array Size iMsg increased to 9999, for reduced VVM Version in General_CP"
"				task c_coupl Bugfix Basisupdate 01: counter MOD 32768 calculation IF536 - IF544 "
"  V4.09.0 BETA	28.11.2019	lettenb. FSM man.test functions with ramp, protection test mapping "
"				06.12.2019	Denk	 Operation Locking for additional Touch Panels "
"				03.02.2020	zengerer task c_set	avoid P setpoint switching with 0mA Value and IN_CU.tP_Set_ExtAI_Norm.GoodQual "
"	BETA   V4.9.0 task c_set 	avoid P setpoint switching with 0mA Value and IN_CU.tP_Set_ExtAI_Norm.GoodQual "
"	UPDATE V4.10.0	03.12.2020	Zengerer MaintenanceCount reset interlock to IN_CU.iCnt_Starts "
"   				27.01.2021  Denk, Bus diagnosis arrays enlarged to 512 (send) and 32 (receive) "
"   				12.03.2021  Zengerer, add file 'CustomizedSpareRegulars' into 'Documents' "
"	UPDATE V4.10.1	xx.08.2021	Zengerer, Gruber Analog Speed Set korr. #530    "
" 								DO NOT USE the IN_CU.tCustDigOut declaration of tCustDigOut anymore! This LEGACY DATA POINT is sheduled to be removed"
"	UPDATE V4.11.0	11.06.2021	Schmid, missing CU vvm mappings for oil supply monitoring added "
"  					30.08.2021  Keller, frequency droop power setpoint (Bus, AI)"
"					24.11.2021 	Zengerer, Heim New predefined linear scaling blocks for plant specific purpose, usage defined hardcodede at time of sw generation.	"
"					17.12.2021 	Schmid, buffer battery check extension"
"	UPDATE V4.11.1	14.02.2022	Schmid, new TC cooling/lubrication table + control battery check supply monitoring mod"
"	UPDATE V4.11.2	23.02.2022	Schmid, +M control battery check option removed - covered by buffer battery check (coordinated execution with starter battery check required)"
"	UPDATE V4.12.0	06.07.2022	Zengerer additional vvm entrys for issue #828 "
"					26.08.2022	Zengerer IF626 Pos_GM_Set_Norm ChangedScaling from V4.12 on -> issue #810 "
"					11.11.2022	Zengerer new IF to GT for customized alarm bits on analog gas pressure sensor "
"					22.12.2022	Zengerer cleanup UniAnaIn, UniDigIn legacy code declarations "
"	UPDATE V4.13.0	22.08.2023	Zengerer remove outdated IN_CU.tCustDigOut (see UPDATE V4.10.1 also) "
"					07.12.2023	Zengerer speed setpoint limitin acc. to issue #1106 "
"					24.08.2023	Zengerer remove ALL IN_CU.bMsgxxxx single bits and replace by array (Issue #1033) "
"                   16.10.2023  Bachler  add IN_CU.bOtherGeneratorsInLSL for bumpless transition to LSL "
"					08.11.2023	Tinello	 bus signal for stopping external EO refill pump"
"					29.11.2023	Goenczi	 New interface variables to other modules"
"					08.12.2023	Denk	 Customer bus coupling with OPC UA"
"	UPDATE V4.14.0 	25.11.2024	Zengerer new IF536 to IF544 handling options with Para.iOpt_Compatible_OpHoursFormat "
"					28.11.2024  Astner   Added IO Mapping to the Plant Communication for customized IOs "
"					29.11.2024	Zengerer new interface for customized EO_FreshOilPump and EO_WasteOilPump DOs"
"					05.03.2025	Denk	 Bugfix, rP_Set_OpcUa wrong datatype #1818 "
"	</Info>"
""
"	<Customized LastModified='4.14.00.0?'>	"
"	See changelog in file 'aeprot'"
"	</Customized>	"
""
"</MODULEFUNCTION>"
;
"</META>"
```

### module_Cust_ORDER.typ - Declare ORDER SPECIFIC DATATYPES in this file
```iecst
(********************************************************************
 * COPYRIGHT -- INNIO Company
 ********************************************************************
 * Package: Customized_Pkg
 * File: module_Cust_ORDER.typ
 * Author: Zengerer
 * Created: Oct. 30, 2012
 ********************************************************************
 * DECLARE PLANT SPECIFIC DATA TYPES HERE, for package Customized_Pkg
 *     (ADD ELEMENTS FOR USE ON ONLY THIS SPECIFIC PLANT HERE)
 ********************************************************************)

TYPE
	IN_Cust_Plant_Struct : 	STRUCT
		ReplaceMeWithYourVariableName : BOOL;
		rCA_IgnP_CylOffset_MDE : ARRAY[0..24]OF REAL; (*Zylinder Z�ndzeitpunktverstellung �ber PUMA*)
		bCA_IgnP_CylOffset_Active_MDE : BOOL; (*Zylinder Z�ndzeitpunktverstellung �ber PUMA aktiv*)
		bCA_IgnP_ActiveMDE : BOOL; (*Aktivierung externe ZZP Regelung �ber PUMA, kommt �ber Visu-Button*)
		bMsg7000 : BOOL; (*OPC-Verbindung zum Pr�fstand ist unterbrochen*)
		rCust_From_PUMA : ARRAY[0..12]OF REAL;  (*Customized variables from PUMA*)
	END_STRUCT;
	OUT_Cust_Plant_Struct : 	STRUCT
		ReplaceMeWithYourVariableName : BOOL;
	END_STRUCT;
	PARA_Cust_Plant_Struct : 	STRUCT
		ReplaceMeWithYourVariableName : BOOL;
	END_STRUCT;
	Vis2MM_Plant_Struct : 	STRUCT
		ReplaceMeWithYourVariableName : BOOL;
	END_STRUCT;
	MM2Vis_Plant_Struct : 	STRUCT
		ReplaceMeWithYourVariableName : BOOL;
		bAirInFan_OutputHWFault : ARRAY[0..3]OF BOOL;
		rAirInFan_Speed : ARRAY[0..3]OF REAL;
		rAirInFan_InputSpeed : ARRAY[0..3]OF REAL;
		rDumpRadiator_Speed : ARRAY[0..3]OF REAL;
		rDumpRadiator_InputSpeed : ARRAY[0..3]OF REAL;
		bAirInFan_DisEngSpeedHigh : ARRAY[0..3]OF BOOL;
		bAirInFan_EngSpeedLow : ARRAY[0..3]OF BOOL;
		bAirInFan_SensorPowerFault : ARRAY[0..3]OF BOOL;
		bAirInFan_SensorPowerHigh : ARRAY[0..3]OF BOOL;
		bAirInFan_SensorPowerLow : ARRAY[0..3]OF BOOL;
		bAirInFan_InputPowerFault : ARRAY[0..3]OF BOOL;
		bAirInFan_InputPowerHigh : ARRAY[0..3]OF BOOL;
		bAirInFan_InputPowerLow : ARRAY[0..3]OF BOOL;
		bAirInFan_ClutchOutputFault : ARRAY[0..3]OF BOOL;
		bAirInFan_ClutchOutputOpen : ARRAY[0..3]OF BOOL;
		bAirInFan_ClutchOutputShort : ARRAY[0..3]OF BOOL;
		bAirInFan_EngineRPMFault : ARRAY[0..3]OF BOOL;
		bAirInFan_APPFault : ARRAY[0..3]OF BOOL;
		bAirInFan_InputSpeedError : ARRAY[0..3]OF BOOL;
		bAirInFan_APTFault : ARRAY[0..3]OF BOOL;
		bAirInFan_OutHardwareFault : ARRAY[0..3]OF BOOL;
		bAirInFan_FanSpeedError : ARRAY[0..3]OF BOOL;
		bAirInFan_ExcessFanSpeed : ARRAY[0..3]OF BOOL;
		bAirInFan_NoFanSpeed : ARRAY[0..3]OF BOOL;
		bAirInFan_FanSpeedPinFault : ARRAY[0..3]OF BOOL;
		bAirInFan_SPN2978InputFault : ARRAY[0..3]OF BOOL;
		bAirInFan_InputSpeedGThanM : ARRAY[0..3]OF BOOL;
		bAirInFan_FanCmdGThanMax : ARRAY[0..3]OF BOOL;
		bAirInFan_FanCmdLThanMITS : ARRAY[0..3]OF BOOL;
		bAirInFan_FanCmdLThanMICS : ARRAY[0..3]OF BOOL;
		bDumpRadiator_OutputHWFault : ARRAY[0..3]OF BOOL;
		bDumpRadiator_DisEngSpeedHigh : ARRAY[0..3]OF BOOL;
		bDumpRadiator_EngSpeedLow : ARRAY[0..3]OF BOOL;
		bDumpRadiator_SensorPowerFault : ARRAY[0..3]OF BOOL;
		bDumpRadiator_SensorPowerHigh : ARRAY[0..3]OF BOOL;
		bDumpRadiator_SensorPowerLow : ARRAY[0..3]OF BOOL;
		bDumpRadiator_InputPowerFault : ARRAY[0..3]OF BOOL;
		bDumpRadiator_InputPowerHigh : ARRAY[0..3]OF BOOL;
		bDumpRadiator_InputPowerLow : ARRAY[0..3]OF BOOL;
		bDumpRadiator_ClutchOutputFault : ARRAY[0..3]OF BOOL;
		bDumpRadiator_ClutchOutputOpen : ARRAY[0..3]OF BOOL;
		bDumpRadiator_ClutchOutputShort : ARRAY[0..3]OF BOOL;
		bDumpRadiator_EngineRPMFault : ARRAY[0..3]OF BOOL;
		bDumpRadiator_APPFault : ARRAY[0..3]OF BOOL;
		bDumpRadiator_InputSpeedError : ARRAY[0..3]OF BOOL;
		bDumpRadiator_APTFault : ARRAY[0..3]OF BOOL;
		bDumpRadiator_OutHardwareFault : ARRAY[0..3]OF BOOL;
		bDumpRadiator_FanSpeedError : ARRAY[0..3]OF BOOL;
		bDumpRadiator_ExcessFanSpeed : ARRAY[0..3]OF BOOL;
		bDumpRadiator_NoFanSpeed : ARRAY[0..3]OF BOOL;
		bDumpRadiator_FanSpeedPinFault : ARRAY[0..3]OF BOOL;
		bDumpRadiator_SPN2978InputFault : ARRAY[0..3]OF BOOL;
		bDumpRadiator_InputSpeedGThanM : ARRAY[0..3]OF BOOL;
		bDumpRadiator_FanCmdGThanMax : ARRAY[0..3]OF BOOL;
		bDumpRadiator_FanCmdLThanMITS : ARRAY[0..3]OF BOOL;
		bDumpRadiator_FanCmdLThanMICS : ARRAY[0..3]OF BOOL;
		bDumpRadiator_WarningMsg : ARRAY[0..3]OF BOOL;
		bAirInFan_WarningMsg : ARRAY[0..3]OF BOOL;
		bDumpRadiatorCAN : ARRAY[0..3]OF BOOL;
		bAirInFanCAN : ARRAY[0..3]OF BOOL;
		bAirInFanRUN : ARRAY[0..3]OF BOOL;
		bDumpRadiatorRUN : ARRAY[0..3]OF BOOL;
		bDumpRadiator_CANWarningMsg : BOOL;
		bAirInFan_CANWarningMsg : BOOL;
	END_STRUCT;
END_TYPE
```

### module_Cust_ORDER.var - Declare ORDER SPECIFIC VARIABLES in this file 
```iecst
(*************************************************************************
 * COPYRIGHT -- INNIO Company
 *************************************************************************
 * Package: Customized_Pkg
 * File: module_Cust_ORDER.var
 * Author: Zengerer
 * Created: December 06, 2012
 ***************************************************************************
 *  ADD ORDER SPECIFIC VARIABLES for package Customized here
 ***************************************************************************
 *
 * ToDo:
 * -----
 *  declare your customized variables here
 *
 ***************************************************************************)
VAR
	bAirInFan_WarningMsg : ARRAY[0..3] OF BOOL;
	bDumpRadiator_WarningMsg : ARRAY[0..3] OF BOOL;
	bAirInFanRUN : ARRAY[0..3] OF BOOL := [4(FALSE)];
	bDumpRadiatorRUN : ARRAY[0..3] OF BOOL := [4(FALSE)];
	bAirInFan_CANWarningMsg : BOOL := FALSE;
	bDumpRadiator_CANWarningMsg : BOOL := FALSE;
	bConnectYourBitHere : BOOL;
END_VAR
```
